FUNCTION_BLOCK MBS_ControlOfOutputs
VAR_INPUT
END_VAR
VAR_OUTPUT
END_VAR
VAR
END_VAR

// NETWORK 1

END_FUNCTION_BLOCK

(* stored: Version 1.1.0.1, ProductVersion 3.1.4024.15
   POU MBS_ControlOfOutputs: Id {93582327-2f33-4c51-8890-fde083b6ae8e}, SpecialFunc None *)
